PROGRAM MAIN
VAR
	fbTestModule1 : TestModule_1;
	fbTestModule2 : TestModule_2;
	fbTestModule3,fbTestModule4,fbTestModule5 : TestModule_3;
END_VAR

fbTestModule1();
fbTestModule2();

//fbTestModule1.fbNextStationReleaseClient.bReleasePresent := fbTestModule2.fbNextStationReleaseMaster.bSetRelease;
//fbTestModule2.fbNextStationReleaseMaster.bReleaseAckIn := fbTestModule1.fbNextStationReleaseClient.bReleaseAckOut;

fbTestModule2.fbNextStationReleaseMaster.SetReleaseClient(fbTestModule1.fbNextStationReleaseClient);
fbTestModule3.fbNextStationReleaseHybrid.SetReleaseClient(fbTestModule4.fbNextStationReleaseHybrid);
fbTestModule4.fbNextStationReleaseHybrid.SetReleaseClient(fbTestModule5.fbNextStationReleaseHybrid);

END_PROGRAM

(* stored: Version 1.1.0.1, ProductVersion 3.1.4024.2
   POU MAIN: Id {6d2efa3e-5b18-456f-af17-8d32ae7e29a2}, SpecialFunc None *)
